TYPE DigitalInputBase :
STRUCT
END_STRUCT
END_TYPE

(* stored: Version 1.1.0.1, ProductVersion 3.1.4024.9
   DUT DigitalInputBase: Id {53074244-94d4-0432-2705-e937beb7b4ed} *)
